TYPE CM_Sensor_HMI :
STRUCT
	Auto		: BOOL;
	Manueel		: BOOL;
	Output		: BOOL;
END_STRUCT
END_TYPE

(* stored: Version 1.1.0.1, ProductVersion 3.1.4024.12
   DUT CM_Sensor_HMI: Id {95301212-0090-4532-920b-8e3d16d33827} *)
